// TIA Portal project "HMI05_Garagentor_V15.1" (V15.1)

(* hardware
DEVICE "S71500/ET200MP-Station_1"  S7-1500 station
   slot 0: "Profilschiene_0"  6ES7 590-1***0-0AA0
   slot 1: "PLC_1"  CPU 1511-1 PN  6ES7 511-1AK01-0AB0  V1.8
   slot 2: "AI 8xU/I/RTD/TC ST_1"  AI 8xU/I/RTD/TC ST  6ES7 531-7KF00-0AB0  V2.0
   slot 3: "AI 8xU/I/RTD/TC ST_2"  AI 8xU/I/RTD/TC ST  6ES7 531-7KF00-0AB0  V2.0
   slot 4: "AI 8xU/I/RTD/TC ST_3"  AI 8xU/I/RTD/TC ST  6ES7 531-7KF00-0AB0  V2.0
   slot 5: "AI 8xU/I/RTD/TC ST_4"  AI 8xU/I/RTD/TC ST  6ES7 531-7KF00-0AB0  V2.0
   slot 6: "DI 16x24VDC BA_1"  DI 16x24VDC BA  6ES7 521-1BH10-0AA0  V1.0
DEVICE "HMI_1"  KTP700 Basic PN
   slot 0: "KTP700 Basic PN"  KTP700 Basic PN  6AV2 123-2GB03-0AX0  14.0.1.0
   slot 1: "HMI_RT_1"  KTP700 Basic PN  6AV2 123-2GB03-0AX0  14.0.1.0
   slot 5: "HMI_1.IE_CP_1"  PROFINET Interface  14.0.1.0
      slot 1: "PROFINET Schnittstelle_1"  PROFINET Interface
         slot 1: "Port_1"  Port
*)

// ===== PLC "PLC_1"  CPU 1511-1 PN =====

VAR_GLOBAL   // PLC tag table "Standard-Variablentabelle"
   "tasteHMIEin" AT %M10.0 : Bool;
   "tasteHMIAus" AT %M10.1 : Bool;
   "fuellstand" AT %MW12 : Int;
END_VAR

ORGANIZATION_BLOCK "Main"   // OB1, FBD, ProgramCycle
TITLE = "Main Program Sweep (Cycle)"
{ S7_Optimized_Access := 'TRUE' }
VERSION : 0.1
   VAR_INPUT
      Initial_Call : Bool;   // Initial call of this OB
      Remanence : Bool;   // =True, if remanent data are available
   END_VAR
BEGIN

REGION Network 1
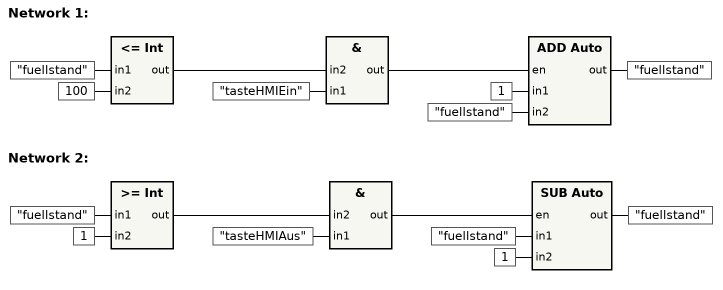
   IF ("fuellstand" <= 100) AND "tasteHMIEin" THEN "fuellstand" := 1 + "fuellstand"; END_IF;
END_REGION

REGION Network 2
   IF ("fuellstand" >= 1) AND "tasteHMIAus" THEN "fuellstand" := "fuellstand" - 1; END_IF;
END_REGION
END_ORGANIZATION_BLOCK

ORGANIZATION_BLOCK "Startup"   // OB100, FBD, Startup
TITLE = "Complete Restart"
{ S7_Optimized_Access := 'TRUE' }
VERSION : 0.1
   VAR_INPUT
      LostRetentive : Bool;   // True if retentive data are lost
      LostRTC : Bool;   // True if date and time are lost
   END_VAR
BEGIN

REGION Network 1
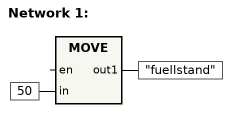
   "fuellstand" := 50;
END_REGION
END_ORGANIZATION_BLOCK

(* ===== HMI "HMI_RT_1" =====
system functions are stored by id; their names below are inferred from use
connection "HMI_Verbindung_1": ETHERNET, SMART_S7_1500_OMS

HMI tags "Standard-Variablentabelle"
   "HMI_TasteEin" : Bool = PLC tasteHMIEin AT %M10.0, 100 ms
   "HMI_TasteAus" : Bool = PLC tasteHMIAus AT %M10.1, 100 ms
   "HMI_fuellst" : Int = PLC fuellstand AT %MW12, 100 ms

text list "Textliste_Bildnamen": 1 'Grundbild'

Template "Vorlage_1" 800x480
   Button "Beenden" at 714,429 size 71x50; TextOff 'Beenden'; PictureOff "ExitRuntime_KTP700_Basic_PN_TR"; PictureOn "ExitRuntime_KTP700_Basic_PN_TR"
      on Release: StopRuntime(0)
   Button "Anmelden" at 614,429 size 71x50; TextOff 'Anmelden'; PictureOff "Login_KTP700_Basic_PN_TR"; PictureOn "Login_KTP700_Basic_PN_TR"
      on Release: function_a2a04561()
   Button "Sprache" at 514,429 size 71x50; TextOff 'Sprache'; PictureOff "ToggleLanguage_KTP700_Basic_PN_TR"; PictureOn "ToggleLanguage_KTP700_Basic_PN_TR"
      on Release: function_fb9197e8(-1)
   Button "Template_Button" at 414,429 size 71x50; TextOff 'Text'
   Button "Template_Button_1" at 314,429 size 71x50; TextOff 'Text'
   Button "Template_Button_2" at 214,429 size 71x50; TextOff 'Text'
   Button "Meldungen" at 114,429 size 71x50; TextOff 'Meldungen'; PictureOff "AlarmDisplay_KTP700_Basic_PN_TR"; PictureOn "AlarmDisplay_KTP700_Basic_PN_TR"
      on Release: function_ef3f5d25("Meldefenster_Nichtquittiert", -1)
   Button "Startbild" at 14,429 size 71x50; TextOff 'Startbild'; PictureOff "NavigateHome_KTP700_Basic_PN_TR"; PictureOn "NavigateHome_KTP700_Basic_PN_TR"
      on Release: ActivateScreen("Grundbild", 0)
   DateTimeField "HmiScreenItemData" at 695,25 size 105x25
   DateTimeField "HmiScreenItemData_1" at 695,0 size 105x25
   GraphicView "Logo" at 0,0 size 91x51; Picture "Logo von HMI_1"

screen "Grundbild" 800x480, template "Vorlage_1"
   TextField "HmiScreenItemData" at 503,375 size 156x25; Text 'Garagentor'
   Button "Schaltfläche_2" at 40,193 size 96x32; TextOff 'Auf'
      on Change: InvertBit("HMI_TasteAus")
   Button "Schaltfläche_1" at 40,258 size 96x32; TextOff 'Zu'
      on Change: InvertBit("HMI_TasteEin")
   Bar "Balken_1" at 221,22 size 550x431; MinimumValue 0; MaximumValue 100
      ProcessValue <- "HMI_fuellst"
   IOField "EA-Feld_1" at 548,66 size 96x32; FormatPattern s999
      ProcessValue <- "HMI_fuellst"
   Circle "Kreis_1" at 713,383 size 48x48
      Appearance <- "HMI_fuellst"
   Circle "Kreis_2" at 705,34 size 48x48
      Appearance <- "HMI_fuellst"
   GraphicView "Grafikanzeige_1" at 2,0 size 196x54; Picture "WH_logo_Just"
*)